KUKA KRL program: TEST1.src, TEST1.dat

--- TEST1.src ---
&ACCESS RVP
&REL 25
DEF TEST1( )
;FOLD INI
    DECL FRAME READY_POS
    DECL FRAME stack_POS
int x
  ;FOLD BASISTECH INI
    GLOBAL INTERRUPT DECL 3 WHEN $STOPMESS==TRUE DO IR_STOPM ( )
    INTERRUPT ON 3
    BAS (#INITMOV,0 )
  ;ENDFOLD (BASISTECH INI)
  ;FOLD USER INI
    ;Make your modifications here

  ;ENDFOLD (USER INI)
;ENDFOLD (INI)

;FOLD PTP HOME Vel=100 % DEFAULT;%{PE}%R 8.3.44,%MKUKATPBASIS,%CMOVE,%VPTP,%P 1:PTP, 2:HOME, 3:, 5:100, 7:DEFAULT
$BWDSTART=FALSE
PDAT_ACT=PDEFAULT
FDAT_ACT=FHOME
BAS(#PTP_PARAMS,100)
$H_POS=XHOME
PTP XHOME
;ENDFOLD
loop
;FOLD PTP pick Vel=100 % PDAT3 Tool[1]:test Base[1]:tesy;%{PE}%R 8.3.44,%MKUKATPBASIS,%CMOVE,%VPTP,%P 1:PTP, 2:pick, 3:, 5:100, 7:PDAT3
$BWDSTART=FALSE
PDAT_ACT=PPDAT3
FDAT_ACT=Fpick
BAS(#PTP_PARAMS,100)
PTP Xpick
;ENDFOLD
;FOLD PTP maduo1 Vel=100 % PDAT1 Tool[1]:test Base[1]:tesy;%{PE}%R 8.3.44,%MKUKATPBASIS,%CMOVE,%VPTP,%P 1:PTP, 2:maduo1, 3:, 5:100, 7:PDAT1
$BWDSTART=FALSE
PDAT_ACT=PPDAT1
FDAT_ACT=Fmaduo1
BAS(#PTP_PARAMS,100)
PTP Xmaduo1
;ENDFOLD
;fold READY_POS
READY_POS=Xmaduo1
READY_POS.X=READY_POS.X+P_POSITION[Tier,Num].X
;READY_POS.Y=READY_POS.Y+P_POSITION[Tier,Num].Y
$BASE=BASE_DATA[1]
FOR X=1 TO 6
$VEL_AXIS[X]=85
$ACC_AXIS[X]=85
ENDFOR
$APO.CPTP=5
ptp READY_POS C_DIS
;endfold
; stack start
;FOLD STACK_POS
stack_POS=Xmaduo1
stack_POS.X=stack_POS.X+P_POSITION[Tier,Num].X
stack_POS.Y=stack_POS.Y+P_POSITION[Tier,Num].Y
stack_POS.Z=stack_POS.Z+P_POSITION[Tier,Num].Z
stack_POS.A=stack_POS.A+P_POSITION[Tier,Num].A
$BASE=BASE_DATA[1]
FOR X=1 TO 6
$VEL_AXIS[X]=85
$ACC_AXIS[X]=85
ENDFOR
$APO.CPTP=5
ptp stack_POS C_DIS
;ENDFOLD
;FOLD COUNT
NUM=NUM+1
if Num>2 then
   Tier=Tier+1
endif
if Tier>2 then
   Tier=1
   NUM=1
exit
;FOLD PULSE 1 'stack finish' State=TRUE Time=3 sec;%{PE}%R 8.2.24,%MKUKATPBASIS,%COUT,%VPULSE,%P 2:1, 3:stack  finish, 5:TRUE, 6:, 8:3
PULSE($OUT[1], TRUE,3)
;ENDFOLD
ENDIF
;ENDFOLD
endloop
;FOLD PTP HOME  Vel= 100 % DEFAULT;%{PE}%MKUKATPBASIS,%CMOVE,%VPTP,%P 1:PTP, 2:HOME, 3:, 5:100, 7:DEFAULT
$BWDSTART = FALSE
PDAT_ACT=PDEFAULT
FDAT_ACT=FHOME
BAS (#PTP_PARAMS,100 )
$H_POS=XHOME
PTP  XHOME
;ENDFOLD

END
def s()
;FOLD PTP maduo2 Vel=100 % PDAT2 Tool[1]:test Base[0];%{PE}%R 8.3.44,%MKUKATPBASIS,%CMOVE,%VPTP,%P 1:PTP, 2:maduo2, 3:, 5:100, 7:PDAT2
$BWDSTART=FALSE
PDAT_ACT=PPDAT2
FDAT_ACT=Fmaduo2
BAS(#PTP_PARAMS,100)
PTP Xmaduo2
;ENDFOLD
end

--- TEST1.dat ---
&ACCESS RVP
&REL 25
DEFDAT  TEST1 PUBLIC
;FOLD EXTERNAL DECLARATIONS;%{PE}%MKUKATPBASIS,%CEXT,%VCOMMON,%P
;FOLD BASISTECH EXT;%{PE}%MKUKATPBASIS,%CEXT,%VEXT,%P
EXT  BAS (BAS_COMMAND  :IN,REAL  :IN )
DECL INT SUCCESS
;ENDFOLD (BASISTECH EXT)
;FOLD USER EXT;%{E}%MKUKATPUSER,%CEXT,%VEXT,%P
;Make here your modifications

;ENDFOLD (USER EXT)
;ENDFOLD (EXTERNAL DECLERATIONS)
DECL BASIS_SUGG_T LAST_BASIS={POINT1[] "pick                    ",POINT2[] "pick                    ",CP_PARAMS[] "CPDAT0                  ",PTP_PARAMS[] "PDAT3                   ",CONT[] "                        ",CP_VEL[] "2.0                     ",PTP_VEL[] "100                     ",SYNC_PARAMS[] "SYNCDAT                 ",SPL_NAME[] "S0                      ",A_PARAMS[] "ADAT0                   "}
DECL E6POS XMADUO1={X 63.7890,Y 141.037537,Z -57.4183273,A 92.7829285,B -2.23925900,C 179.824402,S 2,T 2,E1 0.0,E2 0.0,E3 0.0,E4 0.0,E5 0.0,E6 0.0}
DECL FDAT Fmaduo1={TOOL_NO 1,BASE_NO 1,IPO_FRAME #BASE,POINT2[] " ",TQ_STATE FALSE}
DECL PDAT PPDAT1={VEL 100.000,ACC 100.000,APO_DIST 100.000,GEAR_JERK 50.0000,EXAX_IGN 0}
DECL E6POS XMADUO2={X 457.356689,Y -150.694702,Z 158.085159,A -177.217072,B -2.23925900,C 179.824402,S 2,T 2,E1 0.0,E2 0.0,E3 0.0,E4 0.0,E5 0.0,E6 0.0}
DECL FDAT Fmaduo2={TOOL_NO 1,BASE_NO 0,IPO_FRAME #BASE,POINT2[] " ",TQ_STATE FALSE}
DECL PDAT PPDAT2={VEL 100.000,ACC 100.000,APO_DIST 100.000,GEAR_JERK 50.0000,EXAX_IGN 0}
DECL E6POS XPICK={X 63.6401520,Y 208.102356,Z 29.7364655,A 92.7823792,B -2.24025273,C 179.827744,S 2,T 2,E1 0.0,E2 0.0,E3 0.0,E4 0.0,E5 0.0,E6 0.0}
DECL FDAT Fpick={TOOL_NO 1,BASE_NO 1,IPO_FRAME #BASE,POINT2[] " ",TQ_STATE FALSE}
DECL PDAT PPDAT3={VEL 100.000,ACC 100.000,APO_DIST 100.000,GEAR_JERK 50.0000,EXAX_IGN 0}
ENDDAT
